SUBAPPLICATION Uebung_011g1 (* Numeric Value Input -- multiple IOObservers *)
  (* Standard: 61499-2; Description: Copyright (c) 2023 Meisterschulen am Ostbahnhof This program and the accompanying materials are made available under the terms of the Eclipse Public License 2.0 which is available at https://www.eclipse.org/legal/epl-2.0/ SPDX-License-Identifier: EPL-2.0 *)
  (* Version 1.1, 2026-05-05, Franz Höpfinger, Meisterschulen am Ostbahnhof, multiple IOObservers *)
  (* Version 1.0, 2023-10-23, Franz Höpfinger, Meisterschulen am Ostbahnhof, initial API and implementation and/or initial documentation *)
  PACKAGE Uebungen;
  IMPORT Uebungen::const::UT::DefaultPool::InputNumber_I1;
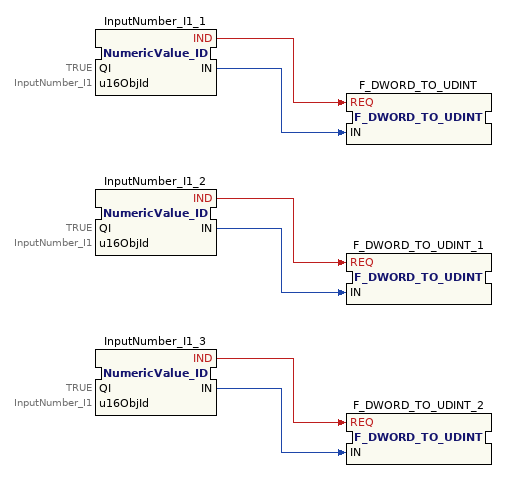
  FBS
    F_DWORD_TO_UDINT : iec61131::conversion::F_DWORD_TO_UDINT;
    InputNumber_I1_1 : isobus::UT::io::NumericValue::NumericValue_ID(QI := TRUE, u16ObjId := InputNumber_I1);
    InputNumber_I1_2 : isobus::UT::io::NumericValue::NumericValue_ID(QI := TRUE, u16ObjId := InputNumber_I1);
    F_DWORD_TO_UDINT_1 : iec61131::conversion::F_DWORD_TO_UDINT;
    InputNumber_I1_3 : isobus::UT::io::NumericValue::NumericValue_ID(QI := TRUE, u16ObjId := InputNumber_I1);
    F_DWORD_TO_UDINT_2 : iec61131::conversion::F_DWORD_TO_UDINT;
  END_FBS
  EVENT_CONNECTIONS
    InputNumber_I1_1.IND TO F_DWORD_TO_UDINT.REQ;
    InputNumber_I1_2.IND TO F_DWORD_TO_UDINT_1.REQ;
    InputNumber_I1_3.IND TO F_DWORD_TO_UDINT_2.REQ;
  END_CONNECTIONS
  DATA_CONNECTIONS
    InputNumber_I1_1.IN TO F_DWORD_TO_UDINT.IN;
    InputNumber_I1_2.IN TO F_DWORD_TO_UDINT_1.IN;
    InputNumber_I1_3.IN TO F_DWORD_TO_UDINT_2.IN;
  END_CONNECTIONS
END_SUBAPPLICATION
